_CFC_ (* Continuous Function Chart, elements in execution order *)
#0 REAL_TO_TIME(SHU6_PV1_P1_ZADER_Z_P1_OTKAZ)
#1 MUL(#0, 1000)
#2 delayFBC_P1 <= #1
#3 AND(#12, SHU6_PV1_1P1_DI7_A)
#4 TON_P1_VKL_Leto:TON(IN: NOT SHU6_PV1_1P1_DO6_VKL, PT: T#5m)
#5 OR(SHU6_PV1_UST_ZIMA, SHU6_PV1_Z_ZAM_SRAB, #4.Q)
#6 TON_P1_OTKL_Leto:TON(IN: SHU6_PV1_1P1_DO6_VKL, PT: T#10s)
#7 AND(SHU6_PV1_UST_LETO, #6.Q)
#8 SR_P1:SR(SET1: #5, RESET: #7)
#9 AND(SHU6_PV1_1P1_DI7_A, SHU6_PV1_1P1_DI4_RUN)
#10 fb_HVACMS_P1:FB_HVACMotor1Speed(eHVACDataSecurityType_Idle, FALSE, TRUE, #8.Q1, eHVACActuatorMode_Auto_BMS, NOT SHU6_PV1_Z_P1_NPIT, #9, NOT SHU6_PV1_Z_P1_OTKAZ, TRUE, TRUE, SHU6_PV1_KV1_DI6, SHU6_PV1_SB, startDelay_P1, stopDelay_P1, delayFBC_P1, feedbPT_P1, delayFBP_P1)
#11 SHU6_PV1_1P1_DO6_VKL <= #10.out 1
#12 >(#10.out 8, 0)
#13 SHU6_PV1_Z_P1_OTKAZ <= #3
#14 SHU6_PV1_1P1_DO8_ALM <= #3
_END_CFC_
END_PROGRAM

(* POU IM/MP1_Upr, CFC *)
PROGRAM MP1_Upr
VAR
	RS_M1: RS;

	startDelay_M1: TIME := T#0s;
	stopDelay_M1: TIME := T#0s;
	delayFBC_M1: TIME := T#30S;
	feedbPT_M1: TIME := T#120s;
	delayFBP_M1: TIME := T#30s;

	fb_HVACMS_M1: FB_HVACMotor1Speed;
	fb_HVACPIDC_M1: FB_HVACPIDCtrl;

	deadRange: REAL := 0.1;
	rKp: REAL := 1;
	tTi: TIME;
	tTv: TIME := T#0s;
	tTd: TIME := T#0s;
	direction: BOOL;
	rYMin: REAL;
	Dint_Ti: DINT;
	set: BOOL;
	reset: BOOL;
	resetContr: BOOL;
	SR_VKL: SR;
	P1_TON: TON;
	PUSK_P1: R_TRIG;
END_VAR
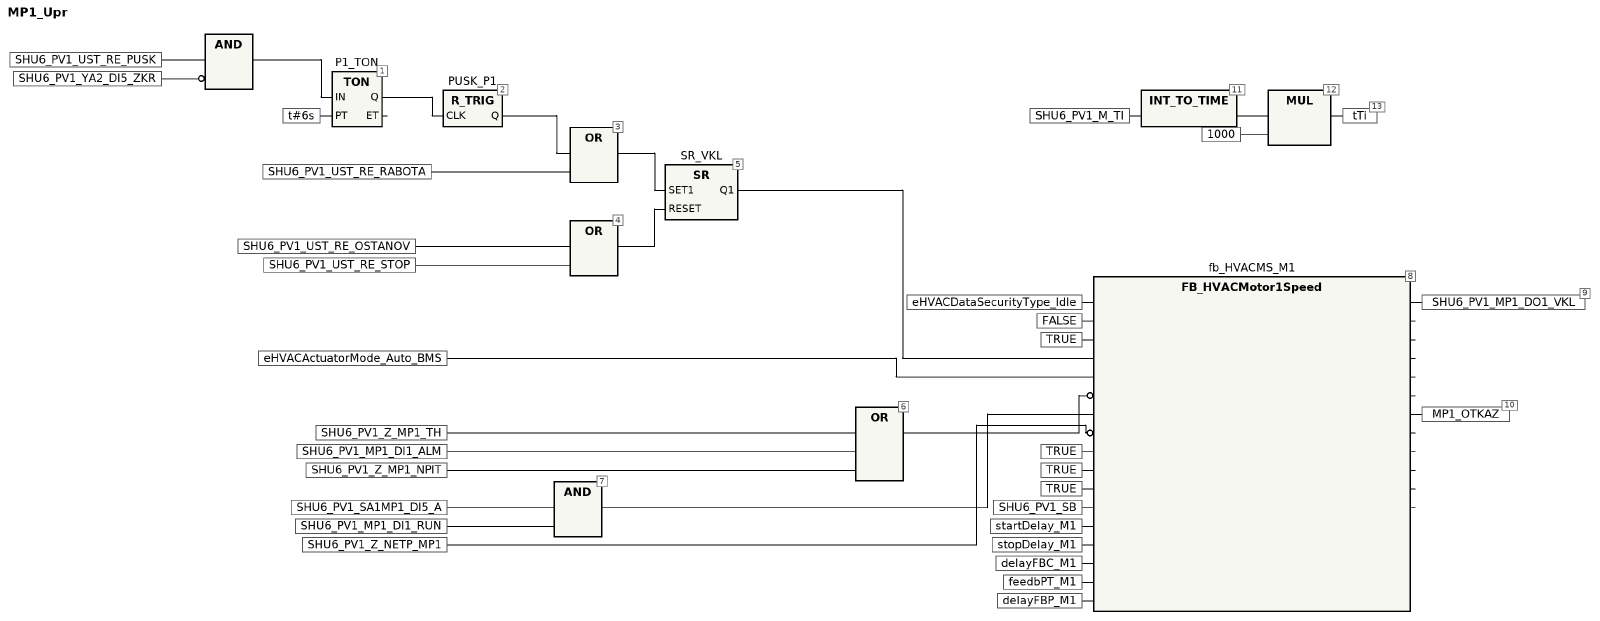
_CFC_ (* Continuous Function Chart, elements in execution order *)
#0 AND(SHU6_PV1_UST_RE_PUSK, NOT SHU6_PV1_YA2_DI5_ZKR)
#1 P1_TON:TON(IN: #0, PT: t#6s)
#2 PUSK_P1:R_TRIG(CLK: #1.Q)
#3 OR(#2.Q, SHU6_PV1_UST_RE_RABOTA)
#4 OR(SHU6_PV1_UST_RE_OSTANOV, SHU6_PV1_UST_RE_STOP)
#5 SR_VKL:SR(SET1: #3, RESET: #4)
#6 OR(SHU6_PV1_Z_MP1_TH, SHU6_PV1_MP1_DI1_ALM, SHU6_PV1_Z_MP1_NPIT)
#7 AND(SHU6_PV1_SA1MP1_DI5_A, SHU6_PV1_MP1_DI1_RUN)
#8 fb_HVACMS_M1:FB_HVACMotor1Speed(eHVACDataSecurityType_Idle, FALSE, TRUE, #5.Q1, eHVACActuatorMode_Auto_BMS, NOT #6, #7, NOT SHU6_PV1_Z_NETP_MP1, TRUE, TRUE, TRUE, SHU6_PV1_SB, startDelay_M1, stopDelay_M1, delayFBC_M1, feedbPT_M1, delayFBP_M1)
#9 SHU6_PV1_MP1_DO1_VKL <= #8.out 1
#10 MP1_OTKAZ <= #8.out 7
#11 INT_TO_TIME(SHU6_PV1_M_TI)
#12 MUL(#11, 1000)
#13 tTi <= #12
_END_CFC_
END_PROGRAM

(* POU IM/MV1_Upr, CFC *)
PROGRAM MV1_Upr
VAR
	RS_M1: RS;

	startDelay_M2: TIME := T#0s;
	stopDelay_M2: TIME := T#0s;
	delayFBC_M2: TIME := T#30S;
	feedbPT_M2: TIME := T#120s;
	delayFBP_M2: TIME := T#30s;

	fb_HVACMS_M2: FB_HVACMotor1Speed;
	fb_HVACPIDC_M1: FB_HVACPIDCtrl;

	deadRange: REAL := 0.1;
	rKp: REAL := 1;
	tTi: TIME;
	tTv: TIME := T#0s;
	tTd: TIME := T#0s;
	direction: BOOL;
	rYMin: REAL;
	Dint_Ti: DINT;
	set: BOOL;
	reset: BOOL;
	resetContr: BOOL;
	SR_VKL: SR;
	mv_1_TON: TON;
END_VAR
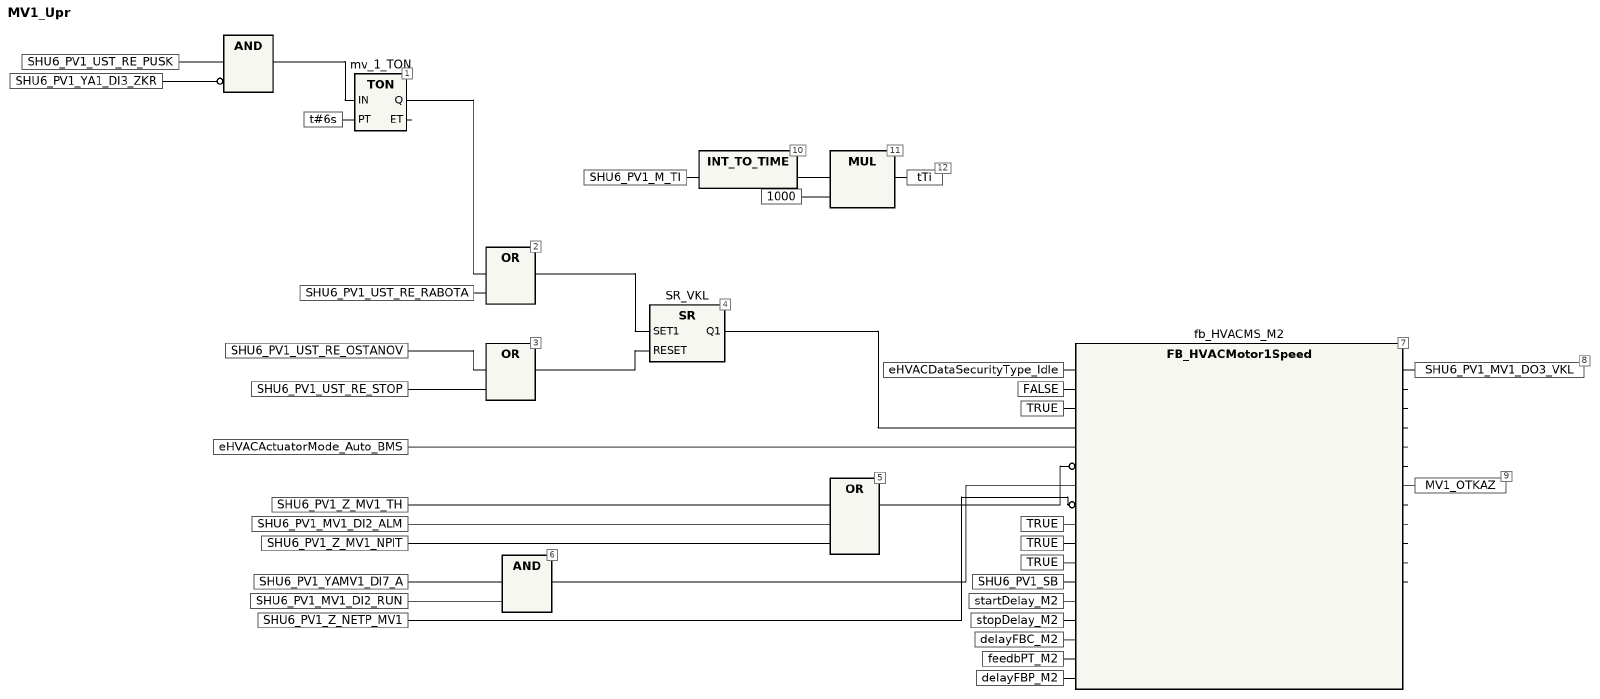
